(* CODESYS project 000TST180401_CodeSys.project

Project tree, tasks and I/O mapping:
  Device : CODESYS Control for Raspberry Pi SL, 3S - Smart Software Solutions GmbH, version 3.5.12.10
    application Application
      libraries: Standard, * (System)
      task MainTask (cyclic, interval 4 ms, priority 1) calls MAIN
      task VISU_TASK (cyclic, interval 100 ms, priority 31) calls VisuElems.Visu_Prg
      DUTs/
        Movitrac B/
          data type ST_Movitrac07B_IN
          data type ST_Movitrac07B_Interface
          data type ST_Movitrac07B_OUT
      GVLs/
        global variables EtherCAT_Variable
        global variables DeviceNET_Variables
        global variables EtherNET_Variables
      POUs/
        program MAIN [ST]: MAIN_IOs, MAIN_MOT
        00_FBs/
          function block FB_Blink [ST]
          function block FB_Movitrac_07B [ST]
        global variables IHM_MAIN
        global variables VAR_MAIN
      VISUs/
        visualisation S00_Principal
      Symbols
    SoftMotion General Axis Pool
    I²C
    SPI
    GPIOs_A_B : GPIOs A/B, 3S - Smart Software Solutions GmbH, version 3.5.11.0
        unmapped channels: digital inputs (GPIO0..GPIO31), digital outputs (GPIO0..GPIO31)
    Onewire
    Camera device
      <Empty>
    EtherCAT_Master : EtherCAT Master, 3S - Smart Software Solutions GmbH, version 3.5.12.20
        settings: NetworkName = 'eth0'; NetworkName = "eth0"; SrcAddress1 = 47143; SrcAddress2 = 3951715331
      EK1100 : EK1100-0030 EtherCAT Coupler (2A E-Bus, 4kV galv. iso.), Beckhoff Automation GmbH & Co. KG, order no. EK1100-0030, version Revision=16#0011001E
          settings: EnableExpertSettings = True; DC sync0 cycletime = 4000; DC sync1 cycletime = 4000
        EL1809 : EL1809 16Ch. Dig. Input 24V, 3ms, Beckhoff Automation GmbH & Co. KG, order no. EL1809, version Revision=16#00120000
            settings: DC sync0 cycletime = 4000; DC sync1 cycletime = 4000
            input  Application.EtherCAT_Variable.EC_DI_00 : BIT  // Input
            input  Application.EtherCAT_Variable.EC_DI_01 : BIT  // Input
            input  Application.EtherCAT_Variable.EC_DI_02 : BIT  // Input
            input  Application.EtherCAT_Variable.EC_DI_03 : BIT  // Input
            input  Application.EtherCAT_Variable.EC_DI_04 : BIT  // Input
            input  Application.EtherCAT_Variable.EC_DI_05 : BIT  // Input
            input  Application.EtherCAT_Variable.EC_DI_06 : BIT  // Input
            input  Application.EtherCAT_Variable.EC_DI_07 : BIT  // Input
            input  Application.EtherCAT_Variable.EC_DI_08 : BIT  // Input
            input  Application.EtherCAT_Variable.EC_DI_09 : BIT  // Input
            input  Application.EtherCAT_Variable.EC_DI_10 : BIT  // Input
            input  Application.EtherCAT_Variable.EC_DI_11 : BIT  // Input
            input  Application.EtherCAT_Variable.EC_DI_12 : BIT  // Input
            input  Application.EtherCAT_Variable.EC_DI_13 : BIT  // Input
            input  Application.EtherCAT_Variable.EC_DI_14 : BIT  // Input
            input  Application.EtherCAT_Variable.EC_DI_15 : BIT  // Input
        EL2809 : EL2809 16Ch. Dig. Output 24V, 0.5A, Beckhoff Automation GmbH & Co. KG, order no. EL2809, version Revision=16#00120000
            settings: DC sync0 cycletime = 4000; DC sync1 cycletime = 4000
            output Application.EtherCAT_Variable.EC_DO_00 : BIT  // Output
            output Application.EtherCAT_Variable.EC_DO_01 : BIT  // Output
            output Application.EtherCAT_Variable.EC_DO_02 : BIT  // Output
            output Application.EtherCAT_Variable.EC_DO_03 : BIT  // Output
            output Application.EtherCAT_Variable.EC_DO_04 : BIT  // Output
            output Application.EtherCAT_Variable.EC_DO_05 : BIT  // Output
            output Application.EtherCAT_Variable.EC_DO_06 : BIT  // Output
            output Application.EtherCAT_Variable.EC_DO_07 : BIT  // Output
            output Application.EtherCAT_Variable.EC_DO_08 : BIT  // Output
            output Application.EtherCAT_Variable.EC_DO_09 : BIT  // Output
            output Application.EtherCAT_Variable.EC_DO_10 : BIT  // Output
            output Application.EtherCAT_Variable.EC_DO_11 : BIT  // Output
            output Application.EtherCAT_Variable.EC_DO_12 : BIT  // Output
            output Application.EtherCAT_Variable.EC_DO_13 : BIT  // Output
            output Application.EtherCAT_Variable.EC_DO_14 : BIT  // Output
            output Application.EtherCAT_Variable.EC_DO_15 : BIT  // Output
        EL3314 : EL3314 4Ch. Ana. Input Thermocouple (TC), Beckhoff Automation GmbH & Co. KG, order no. EL3314, version Revision=16#00170000
            unmapped channels: Status__Underrange, Status__Overrange, Status__Limit 1, Status__Limit 1, Status__Limit 2, Status__Limit 2, Status__Error, ---, ---, ---, ---, ---, ---, ---, Status__TxPDO State, Status__TxPDO Toggle, Value, Status__Underrange, Status__Overrange, Status__Limit 1, Status__Limit 1, Status__Limit 2, Status__Limit 2, Status__Error, ---, ---, ---, ---, ---, ---, ---, Status__TxPDO State, Status__TxPDO Toggle, Value, Status__Underrange, Status__Overrange, Status__Limit 1, Status__Limit 1, Status__Limit 2, Status__Limit 2,
              Status__Error, ---, ---, ---, ---, ---, ---, ---, Status__TxPDO State, Status__TxPDO Toggle, Value, Status__Underrange, Status__Overrange, Status__Limit 1, Status__Limit 1, Status__Limit 2, Status__Limit 2, Status__Error, ---, ---, ---, ---, ---, ---, ---, Status__TxPDO State, Status__TxPDO Toggle, Value
        EL3052 : EL3052 2Ch. Ana. Input 4-20mA, Beckhoff Automation GmbH & Co. KG, order no. EL3052, version Revision=16#00140000
            settings: DC sync0 cycletime = 4000; DC sync1 cycletime = 4000
            unmapped channels: Status__Underrange, Status__Overrange, Status__Limit 1, Status__Limit 1, Status__Limit 2, Status__Limit 2, Status__Error, ---, ---, ---, ---, ---, ---, ---, Status__TxPDO State, Status__TxPDO Toggle, Value, Status__Underrange, Status__Overrange, Status__Limit 1, Status__Limit 1, Status__Limit 2, Status__Limit 2, Status__Error, ---, ---, ---, ---, ---, ---, ---, Status__TxPDO State, Status__TxPDO Toggle, Value
        EL4022 : EL4022 2Ch. Ana. Output 4-20mA, 12bit, Beckhoff Automation GmbH & Co. KG, order no. EL4022, version Revision=16#00140000
            unmapped channels: Analog output, Analog output
        EL6752 : EL6752 DeviceNet Master, Beckhoff Automation GmbH & Co. KG, order no. EL6752, version Revision=16#00140000
            settings: DC sync0 cycletime = 4000; DC sync1 cycletime = 4000
        EL6652 : EL6652 EtherNet/IP Scanner (Master), Beckhoff Automation GmbH & Co. KG, order no. EL6652, version Revision=16#00110000
            settings: DC sync0 cycletime = 4000; DC sync1 cycletime = 4000
      MOVITRAC_FSE24B : MOVITRAC+FSE24B, SEW Eurodrive, order no. MOVITRAC+FSE24B, version Revision=16#00000002
          settings: EnableExpertSettings = True; StationAlias = 1009; Optional = False; DeviceIdenticationADO = 0; DeviceIdenticationMode = 0; DC sync0 cycletime = 4000; DC sync1 cycletime = 4000
          output Application.EC_CTRL_DRIVE_SEW[1] : WORD  // PO 0001
          output Application.EC_CTRL_DRIVE_SEW[2] : WORD  // PO 0002
          output Application.EC_CTRL_DRIVE_SEW[3] : WORD  // PO 0003
          input  Application.EC_STATUS_DRIVE_SEW[1] : WORD  // PI 0001
          input  Application.EC_STATUS_DRIVE_SEW[2] : WORD  // PI 0002
          input  Application.EC_STATUS_DRIVE_SEW[3] : WORD  // PI 0003
  text list GlobalTextList
*)

// Device/Application/DUTs/Movitrac B/ST_Movitrac07B_IN
TYPE ST_Movitrac07B_IN :
STRUCT
	
	MotorEnable					: BOOL; (*Habilita o Motor para Funcionamento na Máquina*)
	InverterStart				: BOOL; (*Bit Gira/Para do Inversor de Frequencia *)
	InverterJog					: BOOL;	(*Bit Executa JOG no motor*)		
	ResetFalhas					: BOOL; (*Bit Reset de Falhas do Inversor de Frequencia *)
	SentidoGiro					: BOOL; (*Bit de Sentido de Giro do Inversor de Frequencia *)
	Velocidade					: REAL; (*Set Point de Velocidade do Inversor de Frequencia*)
	MetrosMinuto				: REAL; (*Set Point de Velocidade em Metros por Minuto do Inversor de Frequencia*)
	NumPolos					: REAL; (*Quantidade de Polos para Calculo de Velocidade*)
	Vel_Min						: REAL; (*Velocidade Mínima do Inversor de Frequencia *)
	Vel_Max						: REAL; (*Velocidade Máxima do Inversor de Frequencia *)
	Proporcao					: REAL; (*Referência de Velocidade proporcional de 0-100%*)
	DiamPrimitivo				: REAL; (*Diametro Primitivo para converter velocidade de m/min para rpm - Usado Apenas em Transportadores*)
	Reducao						: REAL; (*Redução do Redutor para converter velocidade de m/min para rpm - Usado Apenas em Transportadores*)

END_STRUCT
END_TYPE

// Device/Application/DUTs/Movitrac B/ST_Movitrac07B_Interface
TYPE ST_Movitrac07B_Interface :
STRUCT
	
	IN:ST_Movitrac07B_IN;(*Estrutur de entrada para os Inversores de Frequência Movitrac 07B*)
	OUT:ST_Movitrac07B_OUT;(*Estrutur de saída para os Inversores de Frequência Movitrac 07B*)

END_STRUCT
END_TYPE

// Device/Application/DUTs/Movitrac B/ST_Movitrac07B_OUT
TYPE ST_Movitrac07B_OUT :
STRUCT
	
	InverterReady			: BOOL; (*Bit Inversor de Frequencia Habilitado*)
	InverterRunning			: BOOL;	(*Indica Motor girando*)
	ActualDirection			: BOOL;	(*Seleciona Sentido de Giro Horário ou Anti-Horário*)
	InverterFault			: BOOL; (*Bit Genérico de Falha do Drive*)
	VelocidadeAtual			: REAL; (*Velocidade Real do Inversor de Frequencia*)
	CorrenteAtual			: REAL; (*Corrente Atual do Inversor de Frequencia*)
	VelocityRate			: REAL;(*Indica a proporção de 0 - 100% de saida de velocidade*)
	
END_STRUCT
END_TYPE

// Device/Application/GVLs/EtherCAT_Variable
VAR_GLOBAL
	
(*-----------------------------------*)
(* Declaração das Variáveis de I/O's *)
(*-----------------------------------*)
	
	//EtherCAT INPUT
	EC_DI:UINT;
	EC_DI_00:BOOL;
	EC_DI_01:BOOL;
	EC_DI_02:BOOL;
	EC_DI_03:BOOL;
	EC_DI_04:BOOL;
	EC_DI_05:BOOL;
	EC_DI_06:BOOL;
	EC_DI_07:BOOL;
	EC_DI_08:BOOL;
	EC_DI_09:BOOL;
	EC_DI_10:BOOL;
	EC_DI_11:BOOL;
	EC_DI_12:BOOL;
	EC_DI_13:BOOL;
	EC_DI_14:BOOL;
	EC_DI_15:BOOL;
	
	//EtherCAT OUTPUT
	EC_DO:UINT;
	EC_DO_00:BOOL;
	EC_DO_01:BOOL;
	EC_DO_02:BOOL;
	EC_DO_03:BOOL;
	EC_DO_04:BOOL;
	EC_DO_05:BOOL;
	EC_DO_06:BOOL;
	EC_DO_07:BOOL;
	EC_DO_08:BOOL;
	EC_DO_09:BOOL;
	EC_DO_10:BOOL;
	EC_DO_11:BOOL;
	EC_DO_12:BOOL;
	EC_DO_13:BOOL;
	EC_DO_14:BOOL;
	EC_DO_15:BOOL;
	
(*----------------------------------------------------------------*)
(* Declaração das Variáveis de Controle do Inversor de Frequência *)
(*----------------------------------------------------------------*)

(*Control Word*)

	EC_CTRL_DRIVE_SEW :ARRAY [1..3] OF WORD; 		(*Array das Palavras de Controle do Drive*)

(*Status Word*)

	EC_STATUS_DRIVE_SEW :ARRAY [1..3] OF WORD; 		(*Array das Palavras de Status do Drive*)

(*Diagnostic Fault*)

	EC_NETWORK_STATE_DRIVE_SEW :UINT;				(*Status do Drive na Rede*)
	EC_NETWORK_DATA_DRIVE_SEW :BOOL;				(*Disponibilidade dos Dados na Rede "Data Valid = 0" ou "Data Invalid = 1"*)
	
END_VAR

// Device/Application/GVLs/DeviceNET_Variables
VAR_GLOBAL
END_VAR

// Device/Application/GVLs/EtherNET_Variables
VAR_GLOBAL
END_VAR

// Device/Application/POUs/IHM_MAIN
VAR_GLOBAL
END_VAR

// Device/Application/POUs/VAR_MAIN
VAR_GLOBAL

(*Declaração da Estrutura de Controle dos Motores*)

	gDrive_SEW :ST_Movitrac07B_Interface; (*Estrutura de Controle do Inversor de Frequencia*)

END_VAR

// Device/Application/POUs/MAIN
PROGRAM MAIN
VAR
	
(*Declaração da Estrutura de Controle dos Motores*)

	fbDrive_SEW : FB_Movitrac_07B;
	
(*Declaração das Variáveis de uso Geral*)

	Teste01: BOOL;
	Teste02: INT;
	fbBlink: FB_Blink;
	fbRTRIG: R_TRIG;
	
END_VAR

(*Chamada Subrotina de Controle do Espelhamento dos IO's*)
MAIN_IOs ();

(*Chamada Subrotina de Controle dos Motores*)
MAIN_MOT ();

(*Shift Register dos IO's*)
IF (Teste01 OR EC_DI.0) AND NOT EC_DO.15 THEN
	
	fbBlink(Enable:= TRUE, Time_High:= 10, Time_Low:= 10);
	fbRTRIG(CLK:= fbBlink.Blink_Output);
	IF fbRTRIG.Q THEN
		EC_DO := EC_DO*2;
	END_IF;
ELSE
	EC_DO := 1;
END_IF;

ACTION MAIN_IOs:
(*Espelhamento das Saídas Digitais*)
EC_DO_00 := EC_DO.0;
EC_DO_01 := EC_DO.1;
EC_DO_02 := EC_DO.2;
EC_DO_03 := EC_DO.3;
EC_DO_04 := EC_DO.4;
EC_DO_05 := EC_DO.5;
EC_DO_06 := EC_DO.6;
EC_DO_07 := EC_DO.7;
EC_DO_08 := EC_DO.8;
EC_DO_09 := EC_DO.9;
EC_DO_10 := EC_DO.10;
EC_DO_11 := EC_DO.11;
EC_DO_12 := EC_DO.12;
EC_DO_13 := EC_DO.13;
EC_DO_14 := EC_DO.14;
EC_DO_15 := EC_DO.15;

(*Espelhamento das Entradas Digitais*)
EC_DI.0 := EC_DI_00;
EC_DI.1 := EC_DI_01;
EC_DI.2 := EC_DI_02;
EC_DI.3 := EC_DI_03;
EC_DI.4 := EC_DI_04;
EC_DI.5 := EC_DI_05;
EC_DI.6 := EC_DI_06;
EC_DI.7 := EC_DI_07;
EC_DI.8 := EC_DI_08;
EC_DI.9 := EC_DI_09;
EC_DI.10 := EC_DI_10;
EC_DI.11 := EC_DI_11;
EC_DI.12 := EC_DI_12;
EC_DI.13 := EC_DI_13;
EC_DI.14 := EC_DI_14;
EC_DI.15 := EC_DI_15;
END_ACTION

ACTION MAIN_MOT:
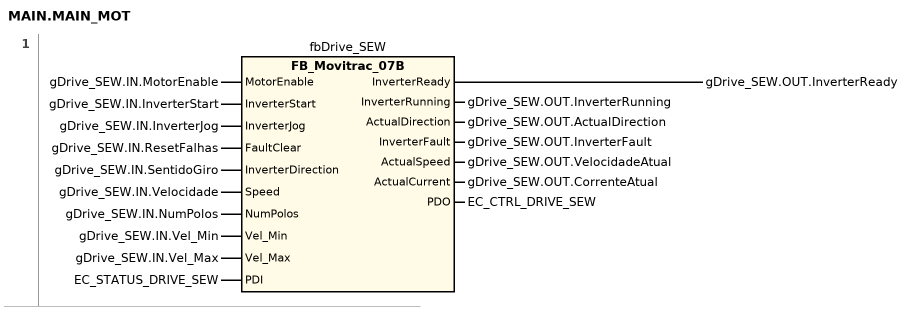
// NETWORK 1
fbDrive_SEW(
    MotorEnable := gDrive_SEW.IN.MotorEnable,
    InverterStart := gDrive_SEW.IN.InverterStart,
    InverterJog := gDrive_SEW.IN.InverterJog,
    FaultClear := gDrive_SEW.IN.ResetFalhas,
    InverterDirection := gDrive_SEW.IN.SentidoGiro,
    Speed := gDrive_SEW.IN.Velocidade,
    NumPolos := gDrive_SEW.IN.NumPolos,
    Vel_Min := gDrive_SEW.IN.Vel_Min,
    Vel_Max := gDrive_SEW.IN.Vel_Max,
    PDI := EC_STATUS_DRIVE_SEW,
    InverterRunning => gDrive_SEW.OUT.InverterRunning,
    ActualDirection => gDrive_SEW.OUT.ActualDirection,
    InverterFault => gDrive_SEW.OUT.InverterFault,
    ActualSpeed => gDrive_SEW.OUT.VelocidadeAtual,
    ActualCurrent => gDrive_SEW.OUT.CorrenteAtual,
    PDO => EC_CTRL_DRIVE_SEW); // FB_Movitrac_07B
gDrive_SEW.OUT.InverterReady := fbDrive_SEW.InverterReady;
END_ACTION

END_PROGRAM

// Device/Application/POUs/00_FBs/FB_Movitrac_07B
FUNCTION_BLOCK FB_Movitrac_07B
VAR_INPUT
	
	MotorEnable					: BOOL; (*Habilita o Funcionamento do Motor*)
	InverterStart				: BOOL; (*Bit Gira/Para do Inversor de Frequencia *)
	InverterJog					: BOOL;	(*Bit Executa JOG no motor*)			
	FaultClear					: BOOL; (*Bit Reset de Falhas do Inversor de Frequencia *)
	InverterDirection			: BOOL; (*Bit de Sentido de Giro do Inversor de Frequencia *)
	Speed						: REAL; (*Set Point de Velocidade do Inversor de Frequencia*)
	NumPolos					: REAL; (*Quantidade de Polos para Calculo de Velocidade*)
	Vel_Min						: REAL; (*Velocidade Mínima do Inversor de Frequencia *)
	Vel_Max						: REAL; (*Velocidade Máxima do Inversor de Frequencia *)
	PDI							: ARRAY [1..3] OF WORD; (*Dados de Entrada do Inversor de Frequência*)
	
END_VAR
VAR_OUTPUT
	
	InverterReady				: BOOL; (*Bit Inversor de Frequencia Habilitado*)
	InverterRunning				: BOOL;	(*Indica Motor girando*)
	ActualDirection				: BOOL;	(*Seleciona Sentido de Giro Horário ou Anti-Horário*)
	InverterFault				: BOOL; (*Bit Genérico de Falha do Drive*)
	ActualSpeed					: REAL; (*Velocidade Real do Inversor de Frequencia*)
	ActualCurrent				: REAL; (*Corrente Atual do Inversor de Frequencia*)
	PDO							: ARRAY [1..3] OF WORD; (*Dados de Saída do Inversor de Frequência*)																																																																																																																																																																																																																																																																																																																																																																																																																																																																																																																																																																																									

END_VAR
VAR
END_VAR

(*Rotinas de Controle do Inversor de Frequência*)

IF MotorEnable THEN //Habilita o Drive
	
(*ROTINAS DE CONTROLE DO DRIVE*)

	(*Habilita o Drive*)
	PDO[1].0 := FALSE;

	(*Start/Stop*)
	IF InverterStart THEN
		PDO[1].1 := TRUE; 	// Normal Stop
		PDO[1].2 := TRUE; 	// Start
	ELSE
		PDO[1].1 := FALSE;	// Normal Stop
		PDO[1].2 := FALSE; 	// Start
	END_IF
	
	(*Clear Fault*)
	PDO[1].6 := FaultClear; //Clear Fault
	
	(*Direction Control*)
	IF InverterDirection THEN
		//Forward Comand CW
		PDO[1].8 := FALSE;
		
		(*Set Point de Velocidade*)
		PDO[2] := REAL_TO_WORD ((Speed/0.2)*-1); //Converte de rpm para unidade de engenharia.
		
	ELSE
		//Reverse Comand CCW
		PDO[1].8 := TRUE;
		
		(*Set Point de Velocidade*)
		PDO[2] := REAL_TO_WORD (Speed/0.2); //Converte de rpm para unidade de engenharia.
		
	END_IF
	
	
(*ROTINAS DE STATUS DO DRIVE*)
	
	(*Drive Ready to Run*)
	InverterReady := PDI[1].1;
	
	(*Drive Running*)
	InverterRunning := PDI[1].0;
	
	(*Inverter Direction*)
	IF (PDI[2] > 0) THEN
		
		ActualDirection := FALSE;
		
	ELSE
		
		ActualDirection := TRUE;
				
	END_IF;
	
	(*Inverter Fault*)
	InverterFault := PDI[1].5;

	(*Feedback de Velocidade Atual*)
	ActualSpeed := ABS((WORD_TO_REAL(PDI[2]))*0.2);
	
	(*Inverter Current*)
	ActualCurrent := PDI[3]*0.01;
	
ELSE
	
	InverterReady := FALSE;
	InverterRunning := FALSE;
	ActualSpeed := 00;
	ActualCurrent := 00;
	PDO[1] := 00;
	PDO[2] := 00;
	PDO[3] := 00;
	
END_IF;

END_FUNCTION_BLOCK

// Device/Application/POUs/00_FBs/FB_Blink
FUNCTION_BLOCK FB_Blink
VAR_INPUT
	
	Enable : BOOL;
	Time_High : REAL;
	Time_Low : REAL;
	
END_VAR
VAR_OUTPUT
	
	Blink_Output : BOOL;
	
END_VAR
VAR
	
	AuxMemoBlink : BOOL;
	fbTON_High: TON;
	fbTON_Low: TON;
	
END_VAR

IF Enable THEN //Habilita a Função BLINK
	
	IF NOT AuxMemoBlink THEN 
			
		Blink_Output:= TRUE; //Aciona a Saída do Bloco
		fbTON_High(IN:= TRUE, PT:= REAL_TO_TIME (Time_High)); //Temporiza a Saída Ligada do Bloco
		fbTON_Low(IN:= FALSE); //Reseta o Temporizador
		
		IF fbTON_High.Q THEN
			AuxMemoBlink := TRUE; //Aciona Memoria Auxiliar que determina que o tempo ligado foi decorrido
		END_IF;
		
	ELSE
		
		Blink_Output:= FALSE; //Desliga a Saída do Bloco
		fbTON_Low(IN:= TRUE, PT:= REAL_TO_TIME (Time_Low)); //Temporiza a Saída Desligada do Bloco
		fbTON_High(IN:= FALSE); //Reseta o Temporizador
		
		IF fbTON_Low.Q THEN
			AuxMemoBlink := FALSE; //Aciona Memoria Auxiliar que determina que o tempo Desligado foi decorrido
		END_IF;
		
	END_IF;
	
ELSE
	
	(*Reset de Todas as Memorias Auxiliares*)
	
	Blink_Output:= FALSE;
	fbTON_Low(IN:= FALSE);
	fbTON_High(IN:= FALSE);

END_IF;

END_FUNCTION_BLOCK

// Device/Application/VISUs/S00_Principal
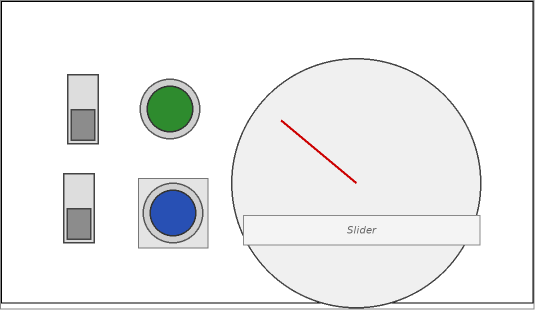
VISUALIZATION S00_Principal  // 535x310
    Rectangle (1,1 532x302)
    Meter180 (231,58 250x250), value: gDrive_SEW.OUT.VelocidadeAtual, style: Meter-Meter180-Gray, scale format: %.1f, scale 0..2000
    Slider (243,215 237x30), variable: gDrive_SEW.IN.Velocidade, scale 0..1800
    DipSwitch (48,74 70x70), variable: gDrive_SEW.IN.MotorEnable, behaviour: TOGGLE, style: Switch-DipSwitch-Gray
    Lamp1 (135,74 70x70), variable: gDrive_SEW.OUT.InverterReady, style: Lamp-Lamp1-Green
    PushSwitchLed (138,178 70x70), variable: gDrive_SEW.IN.InverterStart, behaviour: TOGGLE, style: Switch-PushSwitchLed-Blue
    DipSwitch (44,173 70x70), variable: MAIN.Teste01, behaviour: TOGGLE, style: Switch-DipSwitch-Gray
END_VISUALIZATION
